(* CoDeSys 2.3.9.37 project: tranvia2.pro *)
(* Libraries: Standard.lib 4.10.05 12:14:46, IecSfc.lib 13.4.06 16:51:28 *)

(* Global variable list: Global_Variables *)
VAR_GLOBAL

  (* Entradas *)
   Arranque : BOOL;
   S1 : BOOL;
   S2:BOOL;

   (* Salidas *)
   Sem1CRojo:BOOL :=FALSE;
   Sem1CAmbar:BOOL :=FALSE;
   Sem1CVerde:BOOL :=FALSE;
   Sem1PRojo:BOOL :=FALSE;
   Sem1PVerde:BOOL:=FALSE ;

  Sem2CRojo:BOOL :=FALSE;
   Sem2CAmbar:BOOL :=FALSE;
   Sem2CVerde:BOOL :=FALSE;
   Sem2PRojo:BOOL :=FALSE;
   Sem2PVerde:BOOL:=FALSE ;

   Sem3CRojo:BOOL :=FALSE;
   Sem3CAmbar:BOOL :=FALSE;
   Sem3CVerde:BOOL :=FALSE;
   Sem3PRojo:BOOL :=FALSE;
   Sem3PVerde:BOOL:=FALSE ;

   Sem4CRojo:BOOL :=FALSE;
   Sem4CAmbar:BOOL :=FALSE;
   Sem4CVerde:BOOL :=FALSE;
   Sem4PRojo:BOOL :=FALSE;
   Sem4PVerde:BOOL:=FALSE ;
END_VAR

(* POU PLC_PRG, ST *)
PROGRAM PLC_PRG
VAR
END_VAR
Visualizacion;
END_PROGRAM

(* POU Visualizacion, ST *)
PROGRAM Visualizacion
VAR
   posx: INT :=0;
   posy: INT:= 0;
   ang:INT :=20;
   vectorx : ARRAY[1..56] OF INT :=0,-10,-20,-30,-40,-50,-60,-70,-80,-90,-100,-110,-120,-130,-140,-150,-160,-170,-190,-210,-230,-250,-270,-290,-310,-330,-350,-370,-390,-410,-430,-450,-470,-490,-510,-530,-550,-570,-590,-610,-620,-630,-640,-650,-660,-670,-680,-690,-700,-710,-720,-730,-740,-750,-760,-770;
   vectory : ARRAY[1..56] OF INT:= 21,19,16,10,6,2,-2,-5,-12,-14,-18,-24,-27,-33,-38,-43,-51,-61,-73,-87,-102,-118,-134,-149,-163,-176,-190,-200,-208,-214,-221,-222,-223,-218,-218,-214,-210,-208,-204,-199,-194,-194,-193,-189,-189,-186,-186,-186,-186,-186,-186,-186,-186,-186,-186,-186;
   vectorang : ARRAY[1..56] OF INT:= 220,20,20,20,20,22,22,22,24,25,27,29,30,32,34,35,35,35,37,37,37,37,37,37,34,32,28,24,19,13,4,0,-6,-9,-11,-13,-13,-13,-11,-8,-8,-8,-5,-4,-4,0,0,0,0,0,0,0,0,0,0,0;
   i: INT :=1;

	trenizq: BOOL;
	BotonIzq: BOOL;
	BotonDer: BOOL;
	trender: BOOL;
      cont_vel:INT;
      factor_vel:INT :=1;
	cambiaindice: BOOL;
END_VAR
IF NOT trenizq AND NOT trender THEN
   posx:=10000;
   posy:=10000;
END_IF

IF BotonIzq THEN
   trenizq:=TRUE;
   i:=56;
END_IF

IF BotonDer THEN
   trender:=TRUE;
   i:=1;
END_IF


(*Velocidad del tranvia *)
IF (trenizq OR trender) THEN
  IF  cont_vel=factor_vel THEN
     cont_vel:=1;
     cambiaindice:=TRUE;
  ELSE
     cont_vel:=cont_vel+1;;
     cambiaindice:=FALSE;
 END_IF
END_IF


IF trenizq THEN
   posx:=vectorx[i];
   posy:=vectory[i];
   ang:=vectorang[i];
   IF cambiaindice THEN
         i:=i-1;
   END_IF;
   IF i=0 THEN
      trenizq:=FALSE;
  END_IF
END_IF



IF trender THEN
   posx:=vectorx[i];
   posy:=vectory[i];
   ang:=vectorang[i];
  IF cambiaindice THEN
      i:=i+1;
  END_IF
   IF i=57 THEN
      trender:=FALSE;
  END_IF
END_IF



IF i>=5 AND i<=17 THEN
   S2:=TRUE;
ELSE
   S2:=FALSE;
END_IF;

IF i>=40 AND i<=54 THEN
   S1:=TRUE;
ELSE
   S1:=FALSE;
END_IF;
END_PROGRAM

(* Visualisation Visu
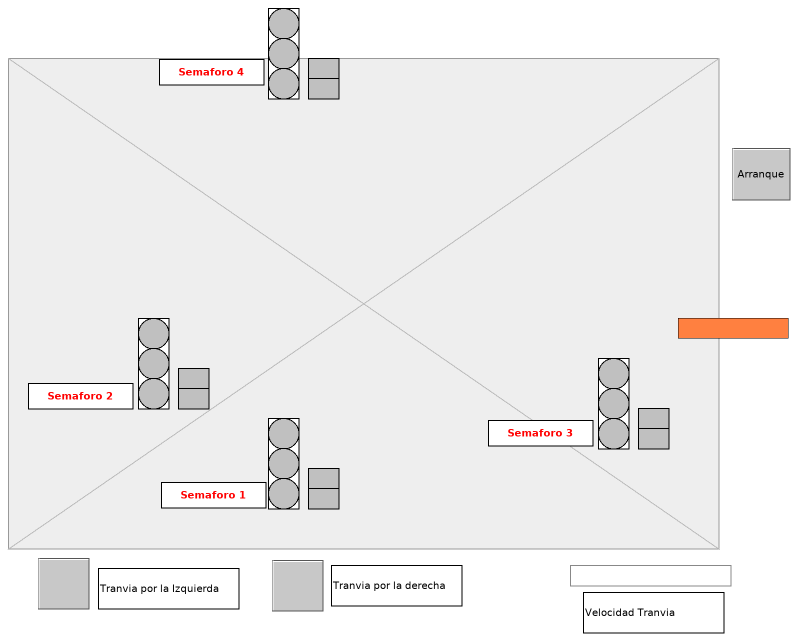
bitmap at (60,50)-(771,541): TRANVIA2.BMP
polygon at (730,310)-(840,330): x offset Visualizacion.posx; y offset Visualizacion.posy; angle Visualizacion.ang
button at (90,550)-(141,601): taps Visualizacion.BotonIzq
button at (324,552)-(375,603): taps Visualizacion.BotonDer
rectangle at (150,560)-(291,601): text "Tranvia por la Izquierda"
rectangle at (383,557)-(514,598): text "Tranvia por la derecha"
rectangle at (635,584)-(776,625): text "Velocidad Tranvia"
ellipse at (320,410)-(351,441): alarm colour if Sem1CRojo
ellipse at (320,440)-(351,471): alarm colour if Sem1CAmbar
ellipse at (320,470)-(351,501): alarm colour if Sem1CVerde
rounded rectangle at (360,460)-(391,481): alarm colour if Sem1PRojo
rounded rectangle at (360,480)-(391,501): alarm colour if Sem1Pverde
ellipse at (650,350)-(681,381): alarm colour if Sem3CRojo
ellipse at (650,380)-(681,411): alarm colour if Sem3CAmbar
ellipse at (650,410)-(681,441): alarm colour if Sem3CVerde
rounded rectangle at (690,400)-(721,421): alarm colour if Sem3PRojo
rounded rectangle at (690,420)-(721,441): alarm colour if Sem3Pverde
ellipse at (190,310)-(221,341): alarm colour if Sem2CRojo
ellipse at (190,340)-(221,371): alarm colour if Sem2CAmbar
ellipse at (190,370)-(221,401): alarm colour if Sem2CVerde
rounded rectangle at (230,360)-(261,381): alarm colour if Sem2PRojo
rounded rectangle at (230,380)-(261,401): alarm colour if Sem2Pverde
ellipse at (320,0)-(351,31): alarm colour if Sem4CRojo
ellipse at (320,30)-(351,61): alarm colour if Sem4CAmbar
ellipse at (320,60)-(351,91): alarm colour if Sem4CVerde
rounded rectangle at (360,50)-(391,71): alarm colour if Sem4PRojo
rounded rectangle at (360,70)-(391,91): alarm colour if Sem4Pverde
rectangle at (80,375)-(185,401): text "Semaforo 2"
rectangle at (213,474)-(318,500): text "Semaforo 1"
rectangle at (540,412)-(645,438): text "Semaforo 3"
rectangle at (211,51)-(316,77): text "Semaforo 4"
button at (784,140)-(842,192): text "Arranque"; toggles Arranque
9 more shapes without text or variables
*)
